// TIA Portal V20 export
TYPE "UDT_Service_ControlBlockMedium"
   STRUCT
      mode : Int := 1;   // Service/Mapping selection
      stepOrder : "UDT_Service_StepOrderRawDataMedium";   // Configuration step order
      "step" : "UDT_Service_StepRawDataMedium";   // Configuration steps
      procedure : "UDT_Service_ProcedureRawDataMedium";   // Configuration procedures
      configurationParameterData : "UDT_Service_ParameterDataMedium";   // Configuration configuration parameters / Configuration parameters
      processValueInData : "UDT_Service_ValueDataMedium";   // Configuration configuration parameters / ProcessIn Values
      processValueOutData : "UDT_Service_ValueDataMedium";   // Configuration configuration parameters / ProcessOut Values
      reportValueData : "UDT_Service_ValueDataMedium";   // Configuration configuration parameters / Report Values
      serviceInteraction : Array[1..30] of DWord;   // Service Interaction Information Variable
      plcGuid : String;   // PLC Guid value stored from the tool, used to find the PLC name changes
      serviceGuid : String;   // Service Guid value stored from the tool, used to find the setup DB name changes
      serviceDbNumber : Int;   // Linked Service IDB number stored from the tool, used to find the service name changes
   END_STRUCT;
END_TYPE
